PROGRAM P_Linked_List_Stack
VAR
	nState 	: BYTE;
	fbStack : FB_Linked_List_Stack;
	
	
	// Init
	bInit_Is_Empty 	: BOOL;
	nInit_Size 		: DINT;
	Init_Top 		: T_DATA_TYPE;
	aInit_Stack 	: ARRAY[1..6] OF T_DATA_TYPE;
	
	// Pust element to stack
	bPush_Is_Empty 	: BOOL;
	nPush_Size 		: DINT;
	Push_Top 		: T_DATA_TYPE;
	Push_Peek		: T_DATA_TYPE;
	aPush_Stack 	: ARRAY[1..6] OF T_DATA_TYPE; 
	
	// Pop element from stack
	bPop_Is_Empty 	: BOOL;
	nPop_Size 		: DINT;
	Pop_Top 		: T_DATA_TYPE;
	aPop_Stack 		: ARRAY[1..6] OF T_DATA_TYPE; 
	
	// Empty Stack
	bEmpty_Is_Empty : BOOL;
	nEmpty_Size 	: DINT;
	Empty_Top 		: T_DATA_TYPE;
	aEmpty_Stack 	: ARRAY[1..6] OF T_DATA_TYPE; 
END_VAR

CASE nState OF
	0: // Init
		bInit_Is_Empty := fbStack.Is_Empty();
		nInit_Size :=  fbStack.Size();
		Init_Top := fbStack.Top();
		fbStack.Show(aInit_Stack);
		
		nState := nState + 1;
		
	1: // Push Element to tack
		fbStack.Push(1);
		fbStack.Push(2);
		fbStack.Push(3);
		fbStack.Push(4);
		fbStack.Push(5);
		bPush_Is_Empty := fbStack.Is_Empty();
		nPush_Size := fbStack.Size();
		Push_Top := fbStack.Top();
		Push_Peek := fbStack.Peek(2);
		fbStack.Show(aPush_Stack);
		
		nState := nState + 1;
	
	2: // Pop elements from stack
		fbStack.Pop();
		fbStack.Pop();
		bPop_Is_Empty := fbStack.Is_Empty();
		nPop_Size := fbStack.Size();
		Pop_Top := fbStack.Top();
		fbStack.Show(aPop_Stack);
		
		nState := nState + 1;
		
	3: // Empty stack
		fbStack.Empty();
		bEmpty_Is_Empty := fbStack.Is_Empty();
		nEmpty_Size := fbStack.Size();
		Empty_Top := fbStack.Top();
		fbStack.Show(aEmpty_Stack);
		
		nState := nState + 1;
END_CASE

END_PROGRAM

(* stored: Version 1.1.0.1, ProductVersion 3.1.4024.4
   POU P_Linked_List_Stack: Id {bc15bfd2-db23-4fc0-ad53-e7306e13d704}, SpecialFunc None *)
